Staubli VAL3: CartesianVel.dtx

public num vx
public num vy
public num vz
public num vrx
public num vry
public num vrz
